LIN {X 0,Y 87.317,Z 374.406,A -85,B 0,C 180,E1 -29312.287,E2 -29312.287} C_VEL
LIN {X 0,Y 96.467,Z 371.337,A -85,B 0,C 180,E1 -29315.588,E2 -29315.588} C_VEL
LIN {X 0,Y 99.391,Z 370.125,A -85,B 0,C 180,E1 -29316.805,E2 -29316.805} C_VEL
LIN {X 0,Y 100.257,Z 369.429,A -85,B 0,C 180,E1 -29319.476,E2 -29319.476} C_VEL
LIN {X 0,Y 101.048,Z 368.656,A -85,B 0,C 180,E1 -29323.841,E2 -29323.841} C_VEL
LIN {X 0,Y 101.506,Z 368.288,A -85,B 0,C 180,E1 -29328.006,E2 -29328.006} C_VEL
LIN {X 0,Y 99.872,Z 368.852,A -85,B 0,C 180,E1 -29330.1,E2 -29330.1} C_VEL
LIN {X 0,Y 92.072,Z 371.42,A -85,B 0,C 180,E1 -29332.851,E2 -29332.851} C_VEL
LIN {X 0,Y 84.521,Z 373.293,A -85,B 0,C 180,E1 -29336.13,E2 -29336.13} C_VEL
LIN {X 0,Y 77.301,Z 374.594,A -85,B 0,C 180,E1 -29340.087,E2 -29340.087} C_VEL
LIN {X 0,Y 69.273,Z 375.318,A -85,B 0,C 180,E1 -29345.814,E2 -29345.814} C_VEL
LIN {X 0,Y 61.992,Z 375.167,A -85,B 0,C 180,E1 -29353.095,E2 -29353.095} C_VEL
LIN {X 0,Y 54.341,Z 373.664,A -85,B 0,C 180,E1 -29365.151,E2 -29365.151} C_VEL
LIN {X 0,Y 49.801,Z 370.828,A -85,B 0,C 180,E1 -29379.102,E2 -29379.102} C_VEL
LIN {X 0,Y 48.399,Z 366.63,A -85,B 0,C 180,E1 -29394.501,E2 -29394.501} C_VEL
LIN {X 0,Y 50.052,Z 360.949,A -85,B 0,C 180,E1 -29409.462,E2 -29409.462} C_VEL
LIN {X 0,Y 53.353,Z 355.031,A -85,B 0,C 180,E1 -29420.53,E2 -29420.53} C_VEL
LIN {X 0,Y 57.912,Z 347.904,A -85,B 0,C 180,E1 -29430.007,E2 -29430.007} C_VEL
LIN {X 0,Y 63.897,Z 338.873,A -85,B 0,C 180,E1 -29438.224,E2 -29438.224} C_VEL
LIN {X 0,Y 70.242,Z 328.519,A -85,B 0,C 180,E1 -29444.491,E2 -29444.491} C_VEL
LIN {X 0,Y 71.313,Z 326.292,A -85,B 0,C 180,E1 -29445.731,E2 -29445.731} C_VEL
LIN {X 0,Y 71.239,Z 323.14,A -85,B 0,C 180,E1 -29448.415,E2 -29448.415} C_VEL
LIN {X 0,Y 70.249,Z 317.78,A -85,B 0,C 180,E1 -29453.595,E2 -29453.595} C_VEL
LIN {X 0,Y 68.353,Z 311.139,A -85,B 0,C 180,E1 -29460.944,E2 -29460.944} C_VEL
LIN {X 0,Y 66.369,Z 305.79,A -85,B 0,C 180,E1 -29468.265,E2 -29468.265} C_VEL
LIN {X 0,Y 64.663,Z 302.071,A -85,B 0,C 180,E1 -29474.897,E2 -29474.897} C_VEL
LIN {X 0,Y 63.575,Z 299.417,A -85,B 0,C 180,E1 -29480.708,E2 -29480.708} C_VEL
LIN {X 0,Y 62.559,Z 298.106,A -85,B 0,C 180,E1 -29485.839,E2 -29485.839} C_VEL
LIN {X 0,Y 61.522,Z 296.631,A -85,B 0,C 180,E1 -29496.064,E2 -29496.064} C_VEL
LIN {X 0,Y 61.542,Z 296.279,A -85,B 0,C 180,E1 -29499.976,E2 -29499.976} C_VEL
LIN {X 0,Y 61.926,Z 296.267,A -85,B 0,C 180,E1 -29506.989,E2 -29506.989} C_VEL
LIN {X 0,Y 62.099,Z 297.173,A -85,B 0,C 180,E1 -29510.532,E2 -29510.532} C_VEL
LIN {X 0,Y 62.252,Z 299.592,A -85,B 0,C 180,E1 -29515.53,E2 -29515.53} C_VEL
LIN {X 0,Y 62.251,Z 302.799,A -85,B 0,C 180,E1 -29520.19,E2 -29520.19} C_VEL
LIN {X 0,Y 63.161,Z 312.359,A -85,B 0,C 180,E1 -29532.44,E2 -29532.44} C_VEL
LIN {X 0,Y 64.224,Z 316.112,A -85,B 0,C 180,E1 -29537.523,E2 -29537.523} C_VEL
LIN {X 0,Y 64.589,Z 321.043,A -85,B 0,C 180,E1 -29542.396,E2 -29542.396} C_VEL
LIN {X 0,Y 64.623,Z 323.854,A -85,B 0,C 180,E1 -29544.935,E2 -29544.935} C_VEL
LIN {X 0,Y 63.02,Z 329.348,A -85,B 0,C 180,E1 -29548.559,E2 -29548.559} C_VEL
LIN {X 0,Y 59.886,Z 337.893,A -85,B 0,C 180,E1 -29554.754,E2 -29554.754} C_VEL
LIN {X 0,Y 58.077,Z 342.441,A -85,B 0,C 180,E1 -29558.641,E2 -29558.641} C_VEL
LIN {X 0,Y 54.908,Z 347.173,A -85,B 0,C 180,E1 -29562.599,E2 -29562.599} C_VEL
LIN {X 0,Y 48.907,Z 355.671,A -85,B 0,C 180,E1 -29572.347,E2 -29572.347} C_VEL
LIN {X 0,Y 44.508,Z 362.423,A -85,B 0,C 180,E1 -29584.253,E2 -29584.253} C_VEL
LIN {X 0,Y 42.222,Z 368.613,A -85,B 0,C 180,E1 -29600.409,E2 -29600.409} C_VEL
LIN {X 0,Y 42.336,Z 371.422,A -85,B 0,C 180,E1 -29609.99,E2 -29609.99} C_VEL
LIN {X 0,Y 42.205,Z 373.519,A -85,B 0,C 180,E1 -29619.576,E2 -29619.576} C_VEL
LIN {X 0,Y 44.947,Z 376.516,A -85,B 0,C 180,E1 -29637.965,E2 -29637.965} C_VEL
LIN {X 0,Y 51.606,Z 378.085,A -85,B 0,C 180,E1 -29652.906,E2 -29652.906} C_VEL
LIN {X 0,Y 61.099,Z 378.262,A -85,B 0,C 180,E1 -29663.616,E2 -29663.616} C_VEL
LIN {X 0,Y 72.168,Z 377.071,A -85,B 0,C 180,E1 -29671.206,E2 -29671.206} C_VEL
LIN {X 0,Y 84.246,Z 374.529,A -85,B 0,C 180,E1 -29676.572,E2 -29676.572} C_VEL
LIN {X 0,Y 93.001,Z 371.88,A -85,B 0,C 180,E1 -29679.331,E2 -29679.331} C_VEL
LIN {X 0,Y 94.006,Z 371.225,A -85,B 0,C 180,E1 -29682.593,E2 -29682.593} C_VEL
LIN {X 0,Y 94.502,Z 370.875,A -85,B 0,C 180,E1 -29685.176,E2 -29685.176} C_VEL
LIN {X 0,Y 94.513,Z 370.771,A -85,B 0,C 180,E1 -29687.103,E2 -29687.103} C_VEL
LIN {X 0,Y 84.658,Z 373.372,A -85,B 0,C 180,E1 -29690.435,E2 -29690.435} C_VEL
LIN {X 0,Y 75.232,Z 375.022,A -85,B 0,C 180,E1 -29694.631,E2 -29694.631} C_VEL
LIN {X 0,Y 66.385,Z 375.756,A -85,B 0,C 180,E1 -29699.991,E2 -29699.991} C_VEL
LIN {X 0,Y 56.825,Z 375.503,A -85,B 0,C 180,E1 -29708.388,E2 -29708.388} C_VEL
LIN {X 0,Y 51.105,Z 374.567,A -85,B 0,C 180,E1 -29715.952,E2 -29715.952} C_VEL
LIN {X 0,Y 45.499,Z 372.585,A -85,B 0,C 180,E1 -29727.59,E2 -29727.59} C_VEL
LIN {X 0,Y 42.078,Z 369.575,A -85,B 0,C 180,E1 -29741.899,E2 -29741.899} C_VEL
LIN {X 0,Y 41.492,Z 364.895,A -85,B 0,C 180,E1 -29759.471,E2 -29759.471} C_VEL
LIN {X 0,Y 43.807,Z 359.491,A -85,B 0,C 180,E1 -29774.223,E2 -29774.223} C_VEL
LIN {X 0,Y 48.484,Z 352.264,A -85,B 0,C 180,E1 -29787.618,E2 -29787.618} C_VEL
LIN {X 0,Y 54.276,Z 344.188,A -85,B 0,C 180,E1 -29797.447,E2 -29797.447} C_VEL
LIN {X 0,Y 60.948,Z 334.614,A -85,B 0,C 180,E1 -29805.044,E2 -29805.044} C_VEL
LIN {X 0,Y 65.289,Z 327.782,A -85,B 0,C 180,E1 -29808.847,E2 -29808.847} C_VEL
LIN {X 0,Y 65.002,Z 323.734,A -85,B 0,C 180,E1 -29813.063,E2 -29813.063} C_VEL
LIN {X 0,Y 64.099,Z 318.961,A -85,B 0,C 180,E1 -29818.722,E2 -29818.722} C_VEL
LIN {X 0,Y 63.264,Z 315.077,A -85,B 0,C 180,E1 -29823.749,E2 -29823.749} C_VEL
LIN {X 0,Y 61.722,Z 310.23,A -85,B 0,C 180,E1 -29831.489,E2 -29831.489} C_VEL
LIN {X 0,Y 60.5,Z 307.092,A -85,B 0,C 180,E1 -29838.283,E2 -29838.283} C_VEL
LIN {X 0,Y 59.754,Z 305.024,A -85,B 0,C 180,E1 -29843.993,E2 -29843.993} C_VEL
LIN {X 0,Y 58.832,Z 303.702,A -85,B 0,C 180,E1 -29851.468,E2 -29851.468} C_VEL
LIN {X 0,Y 58.657,Z 302.901,A -85,B 0,C 180,E1 -29858.946,E2 -29858.946} C_VEL
LIN {X 0,Y 59.011,Z 302.77,A -85,B 0,C 180,E1 -29866.349,E2 -29866.349} C_VEL
LIN {X 0,Y 59.761,Z 303.676,A -85,B 0,C 180,E1 -29873.257,E2 -29873.257} C_VEL
LIN {X 0,Y 60.861,Z 305.478,A -85,B 0,C 180,E1 -29880.01,E2 -29880.01} C_VEL
LIN {X 0,Y 61.892,Z 308.726,A -85,B 0,C 180,E1 -29886.53,E2 -29886.53} C_VEL
LIN {X 0,Y 63.161,Z 312.359,A -85,B 0,C 180,E1 -29892.44,E2 -29892.44} C_VEL
LIN {X 0,Y 63.309,Z 314.892,A -85,B 0,C 180,E1 -29895.107,E2 -29895.107} C_VEL
LIN {X 0,Y 62.621,Z 318.019,A -85,B 0,C 180,E1 -29897.251,E2 -29897.251} C_VEL
LIN {X 0,Y 57.953,Z 329.32,A -85,B 0,C 180,E1 -29903.62,E2 -29903.62} C_VEL
LIN {X 0,Y 54.26,Z 337.976,A -85,B 0,C 180,E1 -29910.324,E2 -29910.324} C_VEL
LIN {X 0,Y 51.65,Z 343.353,A -85,B 0,C 180,E1 -29915.259,E2 -29915.259} C_VEL
LIN {X 0,Y 45.623,Z 351.116,A -85,B 0,C 180,E1 -29922.957,E2 -29922.957} C_VEL
LIN {X 0,Y 39.762,Z 358.714,A -85,B 0,C 180,E1 -29934.927,E2 -29934.927} C_VEL
LIN {X 0,Y 35.693,Z 365.667,A -85,B 0,C 180,E1 -29952.81,E2 -29952.81} C_VEL
LIN {X 0,Y 35.279,Z 370.268,A -85,B 0,C 180,E1 -29969.988,E2 -29969.988} C_VEL
LIN {X 0,Y 35.28,Z 372.523,A -85,B 0,C 180,E1 -29981.479,E2 -29981.479} C_VEL
LIN {X 0,Y 38.831,Z 375.696,A -85,B 0,C 180,E1 -30002.873,E2 -30002.873} C_VEL
LIN {X 0,Y 46.656,Z 377.452,A -85,B 0,C 180,E1 -30018.853,E2 -30018.853} C_VEL
LIN {X 0,Y 57.168,Z 377.88,A -85,B 0,C 180,E1 -30029.365,E2 -30029.365} C_VEL
LIN {X 0,Y 69.016,Z 376.919,A -85,B 0,C 180,E1 -30036.402,E2 -30036.402} C_VEL
LIN {X 0,Y 81.684,Z 374.58,A -85,B 0,C 180,E1 -30041.144,E2 -30041.144} C_VEL
LIN {X 0,Y 86.453,Z 373.375,A -85,B 0,C 180,E1 -30042.462,E2 -30042.462} C_VEL
LIN {X 0,Y 87.432,Z 372.98,A -85,B 0,C 180,E1 -30044.24,E2 -30044.24} C_VEL
LIN {X 0,Y 79.393,Z 374.654,A -85,B 0,C 180,E1 -30046.816,E2 -30046.816} C_VEL
LIN {X 0,Y 71.355,Z 375.716,A -85,B 0,C 180,E1 -30050.008,E2 -30050.008} C_VEL
LIN {X 0,Y 63.586,Z 376.23,A -85,B 0,C 180,E1 -30054.062,E2 -30054.062} C_VEL
LIN {X 0,Y 55.182,Z 376.051,A -85,B 0,C 180,E1 -30059.989,E2 -30059.989} C_VEL
LIN {X 0,Y 47.058,Z 375.007,A -85,B 0,C 180,E1 -30068.576,E2 -30068.576} C_VEL
LIN {X 0,Y 38.66,Z 372.273,A -85,B 0,C 180,E1 -30084.665,E2 -30084.665} C_VEL
LIN {X 0,Y 34.588,Z 368.27,A -85,B 0,C 180,E1 -30104.686,E2 -30104.686} C_VEL
LIN {X 0,Y 34.994,Z 362.86,A -85,B 0,C 180,E1 -30126.33,E2 -30126.33} C_VEL
LIN {X 0,Y 38.425,Z 357.161,A -85,B 0,C 180,E1 -30142.126,E2 -30142.126} C_VEL
LIN {X 0,Y 43.668,Z 350.268,A -85,B 0,C 180,E1 -30154.625,E2 -30154.625} C_VEL
LIN {X 0,Y 50.902,Z 341.037,A -85,B 0,C 180,E1 -30164.925,E2 -30164.925} C_VEL
LIN {X 0,Y 57.725,Z 331.682,A -85,B 0,C 180,E1 -30171.43,E2 -30171.43} C_VEL
LIN {X 0,Y 59.022,Z 329.781,A -85,B 0,C 180,E1 -30172.407,E2 -30172.407} C_VEL
LIN {X 0,Y 59.323,Z 328.38,A -85,B 0,C 180,E1 -30173.764,E2 -30173.764} C_VEL
LIN {X 0,Y 58.885,Z 323.635,A -85,B 0,C 180,E1 -30180.021,E2 -30180.021} C_VEL
LIN {X 0,Y 58.086,Z 318.832,A -85,B 0,C 180,E1 -30187.235,E2 -30187.235} C_VEL
LIN {X 0,Y 57.089,Z 314.386,A -85,B 0,C 180,E1 -30195.721,E2 -30195.721} C_VEL
LIN {X 0,Y 56.45,Z 312.148,A -85,B 0,C 180,E1 -30201.516,E2 -30201.516} C_VEL
LIN {X 0,Y 55.667,Z 310.279,A -85,B 0,C 180,E1 -30209.682,E2 -30209.682} C_VEL
LIN {X 0,Y 55.413,Z 309.398,A -85,B 0,C 180,E1 -30217.648,E2 -30217.648} C_VEL
LIN {X 0,Y 55.747,Z 309.111,A -85,B 0,C 180,E1 -30225.408,E2 -30225.408} C_VEL
LIN {X 0,Y 56.537,Z 310.277,A -85,B 0,C 180,E1 -30234.037,E2 -30234.037} C_VEL
LIN {X 0,Y 57.295,Z 311.993,A -85,B 0,C 180,E1 -30240.011,E2 -30240.011} C_VEL
LIN {X 0,Y 58.569,Z 317.297,A -85,B 0,C 180,E1 -30250.38,E2 -30250.38} C_VEL
LIN {X 0,Y 59.059,Z 319.457,A -85,B 0,C 180,E1 -30253.779,E2 -30253.779} C_VEL
LIN {X 0,Y 59.251,Z 322.629,A -85,B 0,C 180,E1 -30257.617,E2 -30257.617} C_VEL
LIN {X 0,Y 59.1,Z 325.742,A -85,B 0,C 180,E1 -30260.912,E2 -30260.912} C_VEL
LIN {X 0,Y 58.812,Z 327.187,A -85,B 0,C 180,E1 -30262.145,E2 -30262.145} C_VEL
LIN {X 0,Y 57.953,Z 329.32,A -85,B 0,C 180,E1 -30263.62,E2 -30263.62} C_VEL
LIN {X 0,Y 56.361,Z 332.408,A -85,B 0,C 180,E1 -30265.48,E2 -30265.48} C_VEL
LIN {X 0,Y 54.071,Z 335.392,A -85,B 0,C 180,E1 -30266.78,E2 -30266.78} C_VEL
LIN {X 0,Y 45.748,Z 343.816,A -85,B 0,C 180,E1 -30270.523,E2 -30270.523} C_VEL
LIN {X 0,Y 44.912,Z 344.726,A -85,B 0,C 180,E1 -30271.262,E2 -30271.262} C_VEL
LIN {X 0,Y 37.48,Z 353.3,A -85,B 0,C 180,E1 -30281.388,E2 -30281.388} C_VEL
LIN {X 0,Y 31.489,Z 360.367,A -85,B 0,C 180,E1 -30296.069,E2 -30296.069} C_VEL
LIN {X 0,Y 28.332,Z 366.02,A -85,B 0,C 180,E1 -30315.623,E2 -30315.623} C_VEL
LIN {X 0,Y 28.231,Z 369.068,A -85,B 0,C 180,E1 -30329.986,E2 -30329.986} C_VEL
LIN {X 0,Y 28.278,Z 370.151,A -85,B 0,C 180,E1 -30336.009,E2 -30336.009} C_VEL
LIN {X 0,Y 30.058,Z 373.319,A -85,B 0,C 180,E1 -30357.865,E2 -30357.865} C_VEL
LIN {X 0,Y 37.295,Z 376.011,A -85,B 0,C 180,E1 -30378.902,E2 -30378.902} C_VEL
LIN {X 0,Y 47.959,Z 377.292,A -85,B 0,C 180,E1 -30391.534,E2 -30391.534} C_VEL
LIN {X 0,Y 61.342,Z 377.174,A -85,B 0,C 180,E1 -30399.886,E2 -30399.886} C_VEL
LIN {X 0,Y 67.832,Z 376.577,A -85,B 0,C 180,E1 -30402.518,E2 -30402.518} C_VEL
LIN {X 0,Y 70.251,Z 376.192,A -85,B 0,C 180,E1 -30404.089,E2 -30404.089} C_VEL
LIN {X 0,Y 57.097,Z 376.681,A -85,B 0,C 180,E1 -30409.924,E2 -30409.924} C_VEL
LIN {X 0,Y 49.375,Z 376.175,A -85,B 0,C 180,E1 -30415.028,E2 -30415.028} C_VEL
LIN {X 0,Y 42.185,Z 375.131,A -85,B 0,C 180,E1 -30421.935,E2 -30421.935} C_VEL
LIN {X 0,Y 33.127,Z 372.393,A -85,B 0,C 180,E1 -30437.357,E2 -30437.357} C_VEL
LIN {X 0,Y 27.784,Z 368.276,A -85,B 0,C 180,E1 -30460.659,E2 -30460.659} C_VEL
LIN {X 0,Y 27.938,Z 362.707,A -85,B 0,C 180,E1 -30487.855,E2 -30487.855} C_VEL
LIN {X 0,Y 31.978,Z 356.842,A -85,B 0,C 180,E1 -30506.863,E2 -30506.863} C_VEL
LIN {X 0,Y 38.031,Z 349.806,A -85,B 0,C 180,E1 -30520.66,E2 -30520.66} C_VEL
LIN {X 0,Y 45.865,Z 340.757,A -85,B 0,C 180,E1 -30530.851,E2 -30530.851} C_VEL
LIN {X 0,Y 53.47,Z 331.017,A -85,B 0,C 180,E1 -30537.256,E2 -30537.256} C_VEL
LIN {X 0,Y 53.495,Z 327.976,A -85,B 0,C 180,E1 -30541.711,E2 -30541.711} C_VEL
LIN {X 0,Y 53.27,Z 324.37,A -85,B 0,C 180,E1 -30547.686,E2 -30547.686} C_VEL
LIN {X 0,Y 52.875,Z 321.305,A -85,B 0,C 180,E1 -30553.893,E2 -30553.893} C_VEL
LIN {X 0,Y 52.707,Z 319.46,A -85,B 0,C 180,E1 -30558.203,E2 -30558.203} C_VEL
LIN {X 0,Y 52.313,Z 317.665,A -85,B 0,C 180,E1 -30563.726,E2 -30563.726} C_VEL
LIN {X 0,Y 51.826,Z 315.718,A -85,B 0,C 180,E1 -30576.008,E2 -30576.008} C_VEL
LIN {X 0,Y 52.139,Z 315.329,A -85,B 0,C 180,E1 -30584.373,E2 -30584.373} C_VEL
LIN {X 0,Y 52.769,Z 316.057,A -85,B 0,C 180,E1 -30592.358,E2 -30592.358} C_VEL
LIN {X 0,Y 53.299,Z 318.321,A -85,B 0,C 180,E1 -30600.012,E2 -30600.012} C_VEL
LIN {X 0,Y 53.942,Z 322.79,A -85,B 0,C 180,E1 -30609.385,E2 -30609.385} C_VEL
LIN {X 0,Y 54.098,Z 325.165,A -85,B 0,C 180,E1 -30613.152,E2 -30613.152} C_VEL
LIN {X 0,Y 53.761,Z 327.936,A -85,B 0,C 180,E1 -30616.487,E2 -30616.487} C_VEL
LIN {X 0,Y 52.805,Z 330.548,A -85,B 0,C 180,E1 -30618.713,E2 -30618.713} C_VEL
LIN {X 0,Y 48.521,Z 339.012,A -85,B 0,C 180,E1 -30625.77,E2 -30625.77} C_VEL
LIN {X 0,Y 46.462,Z 342.766,A -85,B 0,C 180,E1 -30629.55,E2 -30629.55} C_VEL
LIN {X 0,Y 44.912,Z 344.726,A -85,B 0,C 180,E1 -30631.262,E2 -30631.262} C_VEL
LIN {X 0,Y 41.022,Z 348.554,A -85,B 0,C 180,E1 -30634.449,E2 -30634.449} C_VEL
LIN {X 0,Y 33.505,Z 354.055,A -85,B 0,C 180,E1 -30639.723,E2 -30639.723} C_VEL
LIN {X 0,Y 26.241,Z 359.001,A -85,B 0,C 180,E1 -30648.681,E2 -30648.681} C_VEL
LIN {X 0,Y 23.186,Z 361.878,A -85,B 0,C 180,E1 -30658.38,E2 -30658.38} C_VEL
LIN {X 0,Y 21.183,Z 367.823,A -85,B 0,C 180,E1 -30689.981,E2 -30689.981} C_VEL
LIN {X 0,Y 21.317,Z 368.975,A -85,B 0,C 180,E1 -30698.279,E2 -30698.279} C_VEL
LIN {X 0,Y 24.047,Z 372.305,A -85,B 0,C 180,E1 -30725.749,E2 -30725.749} C_VEL
LIN {X 0,Y 33.069,Z 375.183,A -85,B 0,C 180,E1 -30748.2,E2 -30748.2} C_VEL
LIN {X 0,Y 45.011,Z 376.732,A -85,B 0,C 180,E1 -30759.502,E2 -30759.502} C_VEL
LIN {X 0,Y 51.399,Z 376.979,A -85,B 0,C 180,E1 -30763.136,E2 -30763.136} C_VEL
LIN {X 0,Y 51.939,Z 376.929,A -85,B 0,C 180,E1 -30764.286,E2 -30764.286} C_VEL
LIN {X 0,Y 41.928,Z 375.857,A -85,B 0,C 180,E1 -30770.336,E2 -30770.336} C_VEL
LIN {X 0,Y 32.629,Z 373.878,A -85,B 0,C 180,E1 -30779.981,E2 -30779.981} C_VEL
LIN {X 0,Y 22.978,Z 369.831,A -85,B 0,C 180,E1 -30803.473,E2 -30803.473} C_VEL
LIN {X 0,Y 20.134,Z 364.59,A -85,B 0,C 180,E1 -30838.451,E2 -30838.451} C_VEL
LIN {X 0,Y 22.99,Z 359.601,A -85,B 0,C 180,E1 -30863.653,E2 -30863.653} C_VEL
LIN {X 0,Y 28.62,Z 353.676,A -85,B 0,C 180,E1 -30880.928,E2 -30880.928} C_VEL
LIN {X 0,Y 36.183,Z 346.027,A -85,B 0,C 180,E1 -30892.871,E2 -30892.871} C_VEL
LIN {X 0,Y 44.756,Z 336.597,A -85,B 0,C 180,E1 -30900.697,E2 -30900.697} C_VEL
LIN {X 0,Y 47.403,Z 333.339,A -85,B 0,C 180,E1 -30902.52,E2 -30902.52} C_VEL
LIN {X 0,Y 47.968,Z 332.412,A -85,B 0,C 180,E1 -30903.338,E2 -30903.338} C_VEL
LIN {X 0,Y 48.166,Z 328.719,A -85,B 0,C 180,E1 -30910.35,E2 -30910.35} C_VEL
LIN {X 0,Y 48.162,Z 324.739,A -85,B 0,C 180,E1 -30920.011,E2 -30920.011} C_VEL
LIN {X 0,Y 48.069,Z 323.519,A -85,B 0,C 180,E1 -30924.226,E2 -30924.226} C_VEL
LIN {X 0,Y 47.81,Z 321.986,A -85,B 0,C 180,E1 -30933.847,E2 -30933.847} C_VEL
LIN {X 0,Y 48.174,Z 321.327,A -85,B 0,C 180,E1 -30943.049,E2 -30943.049} C_VEL
LIN {X 0,Y 48.73,Z 321.941,A -85,B 0,C 180,E1 -30951.721,E2 -30951.721} C_VEL
LIN {X 0,Y 48.863,Z 322.992,A -85,B 0,C 180,E1 -30955.889,E2 -30955.889} C_VEL
LIN {X 0,Y 48.981,Z 326.177,A -85,B 0,C 180,E1 -30964.127,E2 -30964.127} C_VEL
LIN {X 0,Y 49.049,Z 328.082,A -85,B 0,C 180,E1 -30968.251,E2 -30968.251} C_VEL
LIN {X 0,Y 48.349,Z 331.155,A -85,B 0,C 180,E1 -30972.476,E2 -30972.476} C_VEL
LIN {X 0,Y 44.109,Z 338.374,A -85,B 0,C 180,E1 -30978.597,E2 -30978.597} C_VEL
LIN {X 0,Y 41.782,Z 342.024,A -85,B 0,C 180,E1 -30982.286,E2 -30982.286} C_VEL
LIN {X 0,Y 40.4,Z 343.847,A -85,B 0,C 180,E1 -30984.025,E2 -30984.025} C_VEL
LIN {X 0,Y 31.885,Z 352.67,A -85,B 0,C 180,E1 -30994.231,E2 -30994.231} C_VEL
LIN {X 0,Y 24.926,Z 359.764,A -85,B 0,C 180,E1 -31010.605,E2 -31010.605} C_VEL
LIN {X 0,Y 23.186,Z 361.878,A -85,B 0,C 180,E1 -31018.38,E2 -31018.38} C_VEL
LIN {X 0,Y 21.618,Z 363.688,A -85,B 0,C 180,E1 -31026.383,E2 -31026.383} C_VEL
LIN {X 0,Y 19.901,Z 365.286,A -85,B 0,C 180,E1 -31035.162,E2 -31035.162} C_VEL
LIN {X 0,Y 17.045,Z 367.916,A -85,B 0,C 180,E1 -31056.962,E2 -31056.962} C_VEL
LIN {X 0,Y 18.401,Z 371.024,A -85,B 0,C 180,E1 -31095.721,E2 -31095.721} C_VEL
LIN {X 0,Y 20.837,Z 371.971,A -85,B 0,C 180,E1 -31104.827,E2 -31104.827} C_VEL
LIN {X 0,Y 29.947,Z 374.333,A -85,B 0,C 180,E1 -31119.801,E2 -31119.801} C_VEL
LIN {X 0,Y 33.254,Z 374.851,A -85,B 0,C 180,E1 -31124.852,E2 -31124.852} C_VEL
LIN {X 0,Y 21.078,Z 371.252,A -85,B 0,C 180,E1 -31140.452,E2 -31140.452} C_VEL
LIN {X 0,Y 14.139,Z 367.27,A -85,B 0,C 180,E1 -31169.753,E2 -31169.753} C_VEL
LIN {X 0,Y 14.323,Z 361.817,A -85,B 0,C 180,E1 -31218.691,E2 -31218.691} C_VEL
LIN {X 0,Y 21.913,Z 354.783,A -85,B 0,C 180,E1 -31248.726,E2 -31248.726} C_VEL
LIN {X 0,Y 31.64,Z 346.143,A -85,B 0,C 180,E1 -31262.151,E2 -31262.151} C_VEL
LIN {X 0,Y 40.804,Z 336.824,A -85,B 0,C 180,E1 -31268.648,E2 -31268.648} C_VEL
LIN {X 0,Y 41.725,Z 335.754,A -85,B 0,C 180,E1 -31269.183,E2 -31269.183} C_VEL
LIN {X 0,Y 42.791,Z 334.027,A -85,B 0,C 180,E1 -31271.08,E2 -31271.08} C_VEL
LIN {X 0,Y 43.146,Z 331.827,A -85,B 0,C 180,E1 -31276.438,E2 -31276.438} C_VEL
LIN {X 0,Y 43.507,Z 329.351,A -85,B 0,C 180,E1 -31283.885,E2 -31283.885} C_VEL
LIN {X 0,Y 43.484,Z 328.116,A -85,B 0,C 180,E1 -31291.013,E2 -31291.013} C_VEL
LIN {X 0,Y 44.001,Z 327.091,A -85,B 0,C 180,E1 -31303.435,E2 -31303.435} C_VEL
LIN {X 0,Y 44.383,Z 327.603,A -85,B 0,C 180,E1 -31310.903,E2 -31310.903} C_VEL
LIN {X 0,Y 44.312,Z 328.783,A -85,B 0,C 180,E1 -31315.466,E2 -31315.466} C_VEL
LIN {X 0,Y 44.001,Z 332.145,A -85,B 0,C 180,E1 -31324.599,E2 -31324.599} C_VEL
LIN {X 0,Y 43.685,Z 333.01,A -85,B 0,C 180,E1 -31325.96,E2 -31325.96} C_VEL
LIN {X 0,Y 39.023,Z 339.785,A -85,B 0,C 180,E1 -31331.9,E2 -31331.9} C_VEL
LIN {X 0,Y 36.42,Z 343.139,A -85,B 0,C 180,E1 -31335.195,E2 -31335.195} C_VEL
LIN {X 0,Y 26.984,Z 352.029,A -85,B 0,C 180,E1 -31344.241,E2 -31344.241} C_VEL
LIN {X 0,Y 18.752,Z 359.161,A -85,B 0,C 180,E1 -31361.414,E2 -31361.414} C_VEL
LIN {X 0,Y 14.092,Z 365.054,A -85,B 0,C 180,E1 -31397.001,E2 -31397.001} C_VEL
LIN {X 0,Y 14.107,Z 366.485,A -85,B 0,C 180,E1 -31409.971,E2 -31409.971} C_VEL
LIN {X 0,Y 14.432,Z 367.805,A -85,B 0,C 180,E1 -31422.92,E2 -31422.92} C_VEL
LIN {X 0,Y 20.837,Z 371.971,A -85,B 0,C 180,E1 -31464.827,E2 -31464.827} C_VEL
LIN {X 0,Y 20.989,Z 372.071,A -85,B 0,C 180,E1 -31467.753,E2 -31467.753} C_VEL
LIN {X 0,Y 19.853,Z 371.726,A -85,B 0,C 180,E1 -31472.935,E2 -31472.935} C_VEL
LIN {X 0,Y 16.702,Z 370.643,A -85,B 0,C 180,E1 -31480.7,E2 -31480.7} C_VEL
LIN {X 0,Y 10.196,Z 367.891,A -85,B 0,C 180,E1 -31498.026,E2 -31498.026} C_VEL
LIN {X 0,Y 6.12,Z 364.906,A -85,B 0,C 180,E1 -31539.378,E2 -31539.378} C_VEL
LIN {X 0,Y 12.26,Z 358.37,A -85,B 0,C 180,E1 -31615.5,E2 -31615.5} C_VEL
LIN {X 0,Y 21.919,Z 351.325,A -85,B 0,C 180,E1 -31629.91,E2 -31629.91} C_VEL
LIN {X 0,Y 31.825,Z 342.844,A -85,B 0,C 180,E1 -31635.883,E2 -31635.883} C_VEL
LIN {X 0,Y 37.771,Z 336.937,A -85,B 0,C 180,E1 -31638.112,E2 -31638.112} C_VEL
LIN {X 0,Y 38.181,Z 335.909,A -85,B 0,C 180,E1 -31640.774,E2 -31640.774} C_VEL
LIN {X 0,Y 38.723,Z 334.231,A -85,B 0,C 180,E1 -31647.031,E2 -31647.031} C_VEL
LIN {X 0,Y 38.928,Z 333.31,A -85,B 0,C 180,E1 -31654.538,E2 -31654.538} C_VEL
LIN {X 0,Y 39.096,Z 332.998,A -85,B 0,C 180,E1 -31658.946,E2 -31658.946} C_VEL
LIN {X 0,Y 39.724,Z 333.055,A -85,B 0,C 180,E1 -31669.826,E2 -31669.826} C_VEL
LIN {X 0,Y 39.174,Z 335.164,A -85,B 0,C 180,E1 -31677.445,E2 -31677.445} C_VEL
LIN {X 0,Y 37.945,Z 337.066,A -85,B 0,C 180,E1 -31680.016,E2 -31680.016} C_VEL
LIN {X 0,Y 33.49,Z 342.372,A -85,B 0,C 180,E1 -31684.427,E2 -31684.427} C_VEL
LIN {X 0,Y 24.929,Z 350.021,A -85,B 0,C 180,E1 -31689.242,E2 -31689.242} C_VEL
LIN {X 0,Y 15.04,Z 357.416,A -85,B 0,C 180,E1 -31700.763,E2 -31700.763} C_VEL
LIN {X 0,Y 7.511,Z 363.37,A -85,B 0,C 180,E1 -31742.045,E2 -31742.045} C_VEL
LIN {X 0,Y 7.039,Z 365.091,A -85,B 0,C 180,E1 -31769.942,E2 -31769.942} C_VEL
LIN {X 0,Y 7.869,Z 366.568,A -85,B 0,C 180,E1 -31796.549,E2 -31796.549} C_VEL
LIN {X 0,Y 15.057,Z 370.078,A -85,B 0,C 180,E1 -31838.916,E2 -31838.916} C_VEL
LIN {X 0,Y 14.439,Z 369.735,A -85,B 0,C 180,E1 -31846.647,E2 -31846.647} C_VEL
LIN {X 0,Y 6.12,Z 364.906,A -85,B 0,C 180,E1 -31899.378,E2 -31899.378} C_VEL
LIN {X 0,Y 6.432,Z 362.266,A -85,B 0,C 180,E1 -31949.135,E2 -31949.135} C_VEL
LIN {X 0,Y 11.98,Z 357.31,A -85,B 0,C 180,E1 -31993.155,E2 -31993.155} C_VEL
LIN {X 0,Y 19.417,Z 351.689,A -85,B 0,C 180,E1 -32006.837,E2 -32006.837} C_VEL
LIN {X 0,Y 24.048,Z 347.981,A -85,B 0,C 180,E1 -32008.619,E2 -32008.619} C_VEL
LIN {X 0,Y 32.883,Z 340.074,A -85,B 0,C 180,E1 -32008.774,E2 -32008.774} C_VEL
LIN {X 0,Y 34.084,Z 338.502,A -85,B 0,C 180,E1 -32015.666,E2 -32015.666} C_VEL
LIN {X 0,Y 34.73,Z 338.302,A -85,B 0,C 180,E1 -32028.343,E2 -32028.343} C_VEL
LIN {X 0,Y 33.644,Z 339.656,A -85,B 0,C 180,E1 -32030.868,E2 -32030.868} C_VEL
LIN {X 0,Y 29.946,Z 343.382,A -85,B 0,C 180,E1 -32032.68,E2 -32032.68} C_VEL
LIN {X 0,Y 19.477,Z 351.919,A -85,B 0,C 180,E1 -32033.047,E2 -32033.047} C_VEL
LIN {X 0,Y 9.736,Z 358.358,A -85,B 0,C 180,E1 -32033.165,E2 -32033.165} C_VEL
LIN {X 0,Y 7.084,Z 359.904,A -85,B 0,C 180,E1 -32033.286,E2 -32033.286} C_VEL
LIN {X 0,Y 5.501,Z 360.634,A -85,B 0,C 180,E1 -32015.773,E2 -32015.773} C_VEL
LIN {X 0,Y 16.44,Z 353.752,A -85,B 0,C 180,E1 -32008.805,E2 -32008.805} C_VEL
LIN {X 0,Y 24.048,Z 347.981,A -85,B 0,C 180,E1 -32008.619,E2 -32008.619} C_VEL
LIN {X 0,Y 27.322,Z 349.523,A -85,B 0,C 180,E1 -32008.598,E2 -32008.598} C_VEL
LIN {X 0,Y 27.322,Z 600,A -85,B 0,C 180,E1 -32008.598,E2 -32008.598} C_VEL
LIN {X 0,Y 27.322,Z 600,A -85,B 0,C 180,E1 -32008.598,E2 -32008.598}

QRS_NEXT_CUT()

QRS_NEXT()
QRS_HOME()

END
